// TwinCAT 3 PLC project PLC1
// ProgramVersion: 3.1.4024.0
// libraries:
//   Tc2_Standard, * (Beckhoff Automation GmbH)
//   Tc2_System, * (Beckhoff Automation GmbH)
//   Tc2_Utilities, * (Beckhoff Automation GmbH)
//   Tc3_Module, * (Beckhoff Automation GmbH)
// project tree:
//   DUTs/ ST_StorageSlot.TcDUT
//   GVLs/ GVL_Config.TcGVL
//   / PlcTask.TcTTO
//   POUs/ FB_SendingData.TcPOU, MAIN.TcPOU
// (motion and I/O tree: see PLC project practice_tdd)
// real-time tasks:
//   TASK PlcTask: cycle T#10ms, priority 20, ADS port 350
//   TASK PlcTask1: cycle T#10ms, priority 21, ADS port 351
//   TASK PlcTask2: cycle T#10ms, priority 22, ADS port 352

CONFIGURATION PLC1
    RESOURCE PLC ON TwinCAT3
        TASK PlcTask(INTERVAL := T#10ms, PRIORITY := 21);
        PROGRAM MAIN WITH PlcTask : MAIN;
    END_RESOURCE
END_CONFIGURATION

// ---- DUTs/ST_StorageSlot.TcDUT
TYPE ST_StorageSlot :
STRUCT
	nStorageId : INT;
	nStorageName : STRING;
	bMaintanence : BOOL;
END_STRUCT
END_TYPE

// ---- GVLs/GVL_Config.TcGVL
{attribute 'qualified_only'}

VAR_GLOBAL
	nNumber : INT := 454;
	arrRack : ARRAY[1..10] OF ST_StorageSlot;
END_VAR

// ---- POUs/MAIN.TcPOU
PROGRAM MAIN
VAR
END_VAR

END_PROGRAM

// ---- POUs/FB_SendingData.TcPOU
FUNCTION_BLOCK FB_SendingData

END_FUNCTION_BLOCK
